TYPE ST_FRConnection :
STRUCT
	_EIPConnectionState AT %I* : UINT;
	_rawIn AT %I*:ARRAY[0..7] OF BYTE;
	_rawOut AT %Q*:ARRAY[0..7] OF BYTE;
END_STRUCT
END_TYPE

(* stored: Version 1.1.0.1, ProductVersion 3.1.4024.15
   DUT ST_FRConnection: Id {3998d349-dbd1-4588-b819-fbc9c6bf61fd} *)
